// TIA Portal project "Proyectogrupal" (V15)

(* hardware
DEVICE "S7-1200 station_1"  S7-1200 Station
   slot 0: "Rack_0"  S7-1200 Rack  Rack  V1.0
   slot 1: "PLC_1"  CPU 1215C AC/DC/Rly  6ES7 215-1BG40-0XB0  V4.2
*)

// ===== PLC "PLC_1"  CPU 1215C AC/DC/Rly =====

VAR_GLOBAL   // PLC tag table "Tabla de variables estándar"
   "Etapa_0" AT %M200.0 : Bool;
   "Etapa_1" AT %M200.1 : Bool;
   "Etapa_2" AT %M200.2 : Bool;
   "Etapa_3" AT %M200.3 : Bool;
   "Etapa_4" AT %M200.4 : Bool;
   "Etapa_5" AT %M200.5 : Bool;
   "Etapa_80" AT %M50.0 : Bool;
   "Etapa_82" AT %M50.2 : Bool;
   "Selector" AT %I0.0 : Bool;
   "PM" AT %I0.1 : Bool;
   "PP" AT %I0.2 : Bool;
   "SH" AT %IW64 : Int;
   "P" AT %IW66 : Int;
   "PV" AT %Q0.0 : Bool;
   "PR" AT %Q0.1 : Bool;
   "Motor_ON" AT %Q0.2 : Bool;
   "Motor_LR" AT %Q0.3 : Bool;
   "Velocidad" AT %MD100 : Real;
   "H" AT %MD800 : Real;
   "AI" AT %QW64 : Int;
   "Clock_Byte" AT %MB0 : Byte;
   "Clock_10Hz" AT %M0.0 : Bool;
   "Clock_5Hz" AT %M0.1 : Bool;
   "Clock_2.5Hz" AT %M0.2 : Bool;
   "Clock_2Hz" AT %M0.3 : Bool;
   "Clock_1.25Hz" AT %M0.4 : Bool;
   "Clock_1Hz" AT %M0.5 : Bool;
   "Clock_0.625Hz" AT %M0.6 : Bool;
   "Clock_0.5Hz" AT %M0.7 : Bool;
   "System_Byte" AT %MB1 : Byte;
   "FirstScan" AT %M1.0 : Bool;
   "DiagStatusUpdate" AT %M1.1 : Bool;
   "AlwaysTRUE" AT %M1.2 : Bool;
   "AlwaysFALSE" AT %M1.3 : Bool;
   "A" AT %MD900 : Real;
   "B(SH)" AT %MD450 : Real;
   "C" AT %MD950 : Real;
   "D(P)" AT %MD475 : Real;
END_VAR

// folder: System blocks/Program resources

DATA_BLOCK "T1_"   // DB2
{ S7_Optimized_Access := 'TRUE' }
AUTHOR : Simatic
FAMILY : IEC
NAME : IEC_TMR
VERSION : 1.0
// stored: InstanceOfName IEC_TIMER
"IEC_TIMER"
BEGIN
END_DATA_BLOCK

// folder: (top level)

FUNCTION "Grafcet_Stop" : Void   // FC1, LAD
{ S7_Optimized_Access := 'TRUE' }
VERSION : 0.1
BEGIN

REGION Network 1
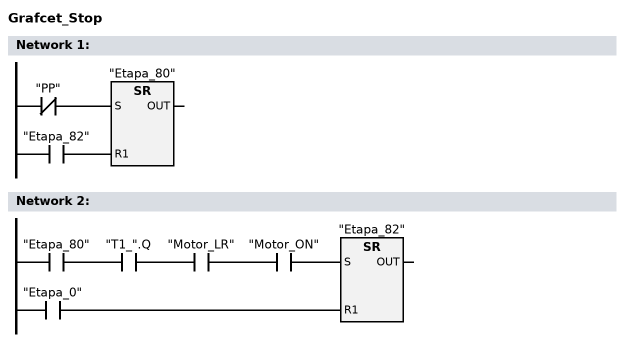
   RUNG wire#powerrail
      I_Contact( "PP" )
      S_SR(operand := "Etapa_80", r1 := wire#w1)
   END_RUNG
   RUNG wire#powerrail
      Contact( "Etapa_82" )
   END_RUNG wire#w1
   // the same network as SCL:
   IF NOT "PP" THEN
       "Etapa_80" := TRUE;   // SR flip-flop
   END_IF;
   IF "Etapa_82" THEN "Etapa_80" := FALSE; END_IF;
END_REGION

REGION Network 2
   RUNG wire#powerrail
      Contact( "Etapa_80" )
      Contact( "T1_".Q )
      Contact( "Motor_LR" )
      Contact( "Motor_ON" )
      S_SR(operand := "Etapa_82", r1 := wire#w1)
   END_RUNG
   RUNG wire#powerrail
      Contact( "Etapa_0" )
   END_RUNG wire#w1
   // the same network as SCL:
   IF "Etapa_80" AND "T1_".Q AND "Motor_LR" AND "Motor_ON" THEN
       "Etapa_82" := TRUE;   // SR flip-flop
   END_IF;
   IF "Etapa_0" THEN "Etapa_82" := FALSE; END_IF;
END_REGION
END_FUNCTION

FUNCTION "Grafcet_Automatico" : Void   // FC2, LAD
{ S7_Optimized_Access := 'TRUE' }
VERSION : 0.1
BEGIN

REGION Network 1
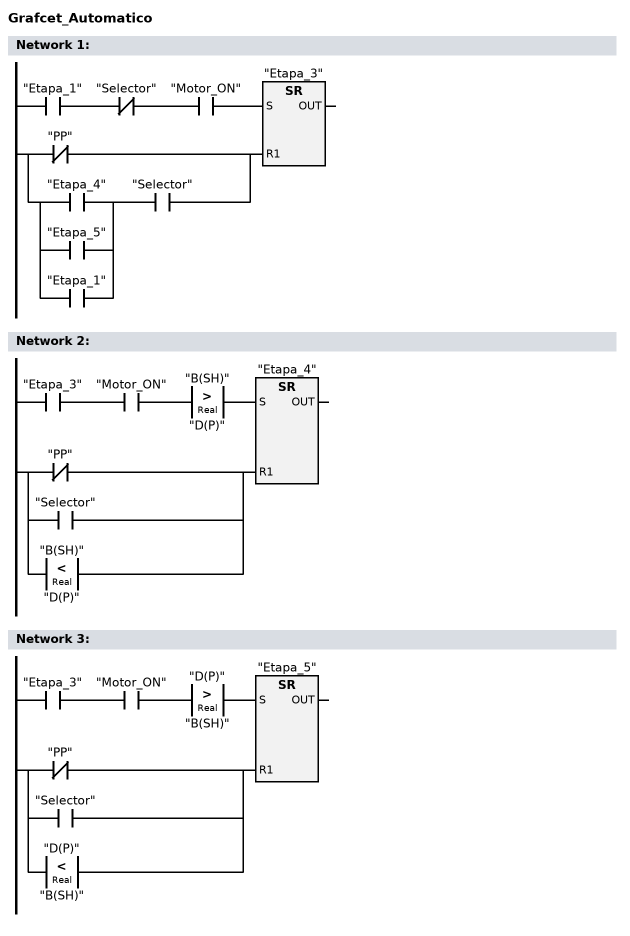
   RUNG wire#powerrail
      Contact( "Etapa_1" )
      I_Contact( "Selector" )
      Contact( "Motor_ON" )
      S_SR(operand := "Etapa_3", r1 := wire#w2)
   END_RUNG
   RUNG wire#powerrail
      I_Contact( "PP" )
   END_RUNG wire#w2
   RUNG wire#powerrail
      Contact( "Etapa_4" )
      wire#w1
      Contact( "Selector" )
   END_RUNG wire#w2
   RUNG wire#powerrail
      Contact( "Etapa_5" )
   END_RUNG wire#w1
   RUNG wire#powerrail
      Contact( "Etapa_1" )
   END_RUNG wire#w1
   // the same network as SCL:
   IF "Etapa_1" AND NOT "Selector" AND "Motor_ON" THEN
       "Etapa_3" := TRUE;   // SR flip-flop
   END_IF;
   IF NOT "PP" OR (("Etapa_4" OR "Etapa_5" OR "Etapa_1") AND "Selector") THEN "Etapa_3" := FALSE; END_IF;
END_REGION

REGION Network 2
   RUNG wire#powerrail
      Contact( "Etapa_3" )
      Contact( "Motor_ON" )
      { S7_Templates := "SrcType := Real" } GT_Contact(in1 := "B(SH)", in2 := "D(P)")
      S_SR(operand := "Etapa_4", r1 := wire#w1)
   END_RUNG
   RUNG wire#powerrail
      I_Contact( "PP" )
   END_RUNG wire#w1
   RUNG wire#powerrail
      Contact( "Selector" )
   END_RUNG wire#w1
   RUNG wire#powerrail
      { S7_Templates := "SrcType := Real" } LT_Contact(in1 := "B(SH)", in2 := "D(P)")
   END_RUNG wire#w1
   // the same network as SCL:
   IF "Etapa_3" AND "Motor_ON" AND ("B(SH)" > "D(P)") THEN
       "Etapa_4" := TRUE;   // SR flip-flop
   END_IF;
   IF NOT "PP" OR "Selector" OR ("B(SH)" < "D(P)") THEN "Etapa_4" := FALSE; END_IF;
END_REGION

REGION Network 3
   RUNG wire#powerrail
      Contact( "Etapa_3" )
      Contact( "Motor_ON" )
      { S7_Templates := "SrcType := Real" } GT_Contact(in1 := "D(P)", in2 := "B(SH)")
      S_SR(operand := "Etapa_5", r1 := wire#w1)
   END_RUNG
   RUNG wire#powerrail
      I_Contact( "PP" )
   END_RUNG wire#w1
   RUNG wire#powerrail
      Contact( "Selector" )
   END_RUNG wire#w1
   RUNG wire#powerrail
      { S7_Templates := "SrcType := Real" } LT_Contact(in1 := "D(P)", in2 := "B(SH)")
   END_RUNG wire#w1
   // the same network as SCL:
   IF "Etapa_3" AND "Motor_ON" AND ("D(P)" > "B(SH)") THEN
       "Etapa_5" := TRUE;   // SR flip-flop
   END_IF;
   IF NOT "PP" OR "Selector" OR ("D(P)" < "B(SH)") THEN "Etapa_5" := FALSE; END_IF;
END_REGION
END_FUNCTION

FUNCTION "Grafcet_Manual" : Void   // FC3, LAD
{ S7_Optimized_Access := 'TRUE' }
VERSION : 0.1
BEGIN

REGION Network 1
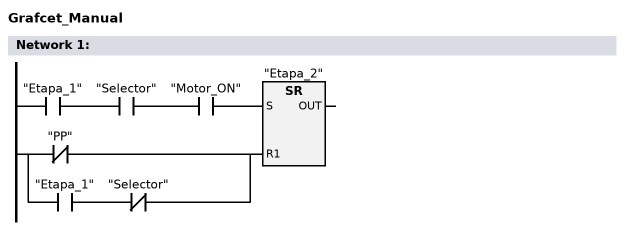
   RUNG wire#powerrail
      Contact( "Etapa_1" )
      Contact( "Selector" )
      Contact( "Motor_ON" )
      S_SR(operand := "Etapa_2", r1 := wire#w1)
   END_RUNG
   RUNG wire#powerrail
      I_Contact( "PP" )
   END_RUNG wire#w1
   RUNG wire#powerrail
      Contact( "Etapa_1" )
      I_Contact( "Selector" )
   END_RUNG wire#w1
   // the same network as SCL:
   IF "Etapa_1" AND "Selector" AND "Motor_ON" THEN
       "Etapa_2" := TRUE;   // SR flip-flop
   END_IF;
   IF NOT "PP" OR ("Etapa_1" AND NOT "Selector") THEN "Etapa_2" := FALSE; END_IF;
END_REGION
END_FUNCTION

FUNCTION "Grafcet_Acciones" : Void   // FC4, LAD
{ S7_Optimized_Access := 'TRUE' }
VERSION : 0.1
BEGIN

REGION Network 1
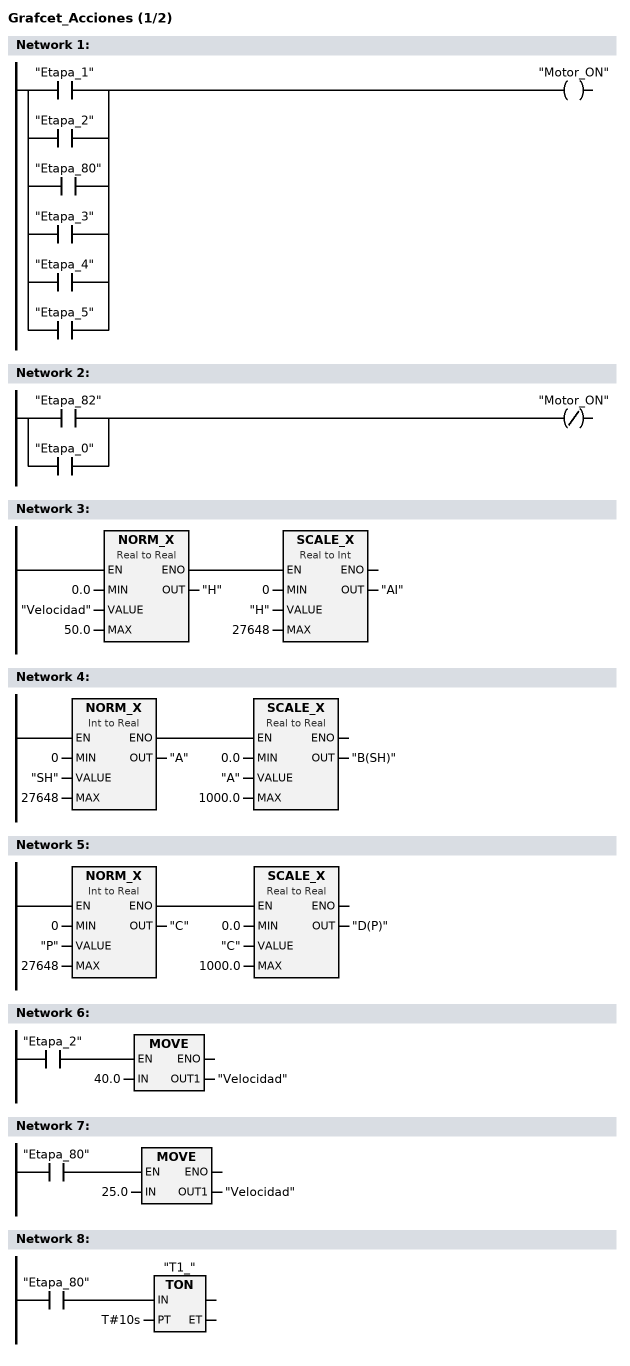
   RUNG wire#powerrail
      Contact( "Etapa_1" )
      wire#w1
      Coil( "Motor_ON" )
   END_RUNG
   RUNG wire#powerrail
      Contact( "Etapa_2" )
   END_RUNG wire#w1
   RUNG wire#powerrail
      Contact( "Etapa_80" )
   END_RUNG wire#w1
   RUNG wire#powerrail
      Contact( "Etapa_3" )
   END_RUNG wire#w1
   RUNG wire#powerrail
      Contact( "Etapa_4" )
   END_RUNG wire#w1
   RUNG wire#powerrail
      Contact( "Etapa_5" )
   END_RUNG wire#w1
   // the same network as SCL:
   "Motor_ON" := "Etapa_1" OR "Etapa_2" OR "Etapa_80" OR "Etapa_3" OR "Etapa_4" OR "Etapa_5";
END_REGION

REGION Network 2
   RUNG wire#powerrail
      Contact( "Etapa_82" )
      wire#w1
      I_Coil( "Motor_ON" )
   END_RUNG
   RUNG wire#powerrail
      Contact( "Etapa_0" )
   END_RUNG wire#w1
   // the same network as SCL:
   "Motor_ON" := NOT ("Etapa_82" OR "Etapa_0");
END_REGION

REGION Network 3
   RUNG wire#powerrail
      { S7_Templates := "[SrcType := Real, DestType := Real]" } Normalize(min := 0.0, value := "Velocidad", max := 50.0, out => "H")
      { S7_Templates := "[SrcType := Real, DestType := Int]" } Scale(min := 0, value := "H", max := 27648, out => "AI")
   END_RUNG
   // the same network as SCL:
   "H" := NORM_X(MIN := 0.0, VALUE := "Velocidad", MAX := 50.0);
   "AI" := SCALE_X(MIN := 0, VALUE := "H", MAX := 27648);
END_REGION

REGION Network 4
   RUNG wire#powerrail
      { S7_Templates := "[SrcType := Int, DestType := Real]" } Normalize(min := 0, value := "SH", max := 27648, out => "A")
      { S7_Templates := "[SrcType := Real, DestType := Real]" } Scale(min := 0.0, value := "A", max := 1000.0, out => "B(SH)")
   END_RUNG
   // the same network as SCL:
   "A" := NORM_X(MIN := 0, VALUE := "SH", MAX := 27648);
   "B(SH)" := SCALE_X(MIN := 0.0, VALUE := "A", MAX := 1000.0);
END_REGION

REGION Network 5
   RUNG wire#powerrail
      { S7_Templates := "[SrcType := Int, DestType := Real]" } Normalize(min := 0, value := "P", max := 27648, out => "C")
      { S7_Templates := "[SrcType := Real, DestType := Real]" } Scale(min := 0.0, value := "C", max := 1000.0, out => "D(P)")
   END_RUNG
   // the same network as SCL:
   "C" := NORM_X(MIN := 0, VALUE := "P", MAX := 27648);
   "D(P)" := SCALE_X(MIN := 0.0, VALUE := "C", MAX := 1000.0);
END_REGION

REGION Network 6
   RUNG wire#powerrail
      Contact( "Etapa_2" )
      Move(in := 40.0, out1 => "Velocidad")
   END_RUNG
   // the same network as SCL:
   IF "Etapa_2" THEN "Velocidad" := 40.0; END_IF;
END_REGION

REGION Network 7
   RUNG wire#powerrail
      Contact( "Etapa_80" )
      Move(in := 25.0, out1 => "Velocidad")
   END_RUNG
   // the same network as SCL:
   IF "Etapa_80" THEN "Velocidad" := 25.0; END_IF;
END_REGION

REGION Network 8
   "T1_".TON(IN := "Etapa_80", PT := T#10s);
END_REGION

REGION Network 9
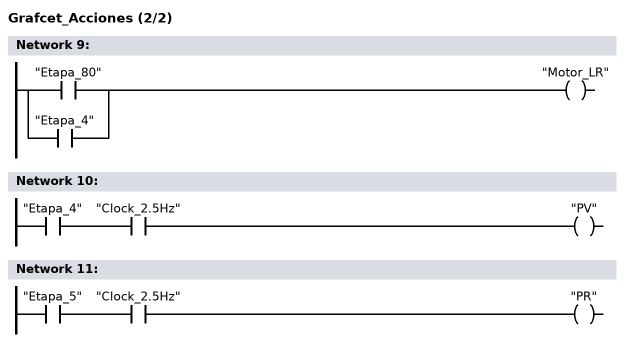
   RUNG wire#powerrail
      Contact( "Etapa_80" )
      wire#w1
      Coil( "Motor_LR" )
   END_RUNG
   RUNG wire#powerrail
      Contact( "Etapa_4" )
   END_RUNG wire#w1
   // the same network as SCL:
   "Motor_LR" := "Etapa_80" OR "Etapa_4";
END_REGION

REGION Network 10
   RUNG wire#powerrail
      Contact( "Etapa_4" )
      Contact( "Clock_2.5Hz" )
      Coil( "PV" )
   END_RUNG
   // the same network as SCL:
   "PV" := "Etapa_4" AND "Clock_2.5Hz";
END_REGION

REGION Network 11
   RUNG wire#powerrail
      Contact( "Etapa_5" )
      Contact( "Clock_2.5Hz" )
      Coil( "PR" )
   END_RUNG
   // the same network as SCL:
   "PR" := "Etapa_5" AND "Clock_2.5Hz";
END_REGION
END_FUNCTION

ORGANIZATION_BLOCK "Main"   // OB1, LAD, ProgramCycle
TITLE = "Main Program Sweep (Cycle)"
{ S7_Optimized_Access := 'TRUE' }
VERSION : 0.1
   VAR_INPUT
      Initial_Call : Bool;   // Initial call of this OB
      Remanence : Bool;   // =True, if remanent data are available
   END_VAR
BEGIN

REGION Network 1
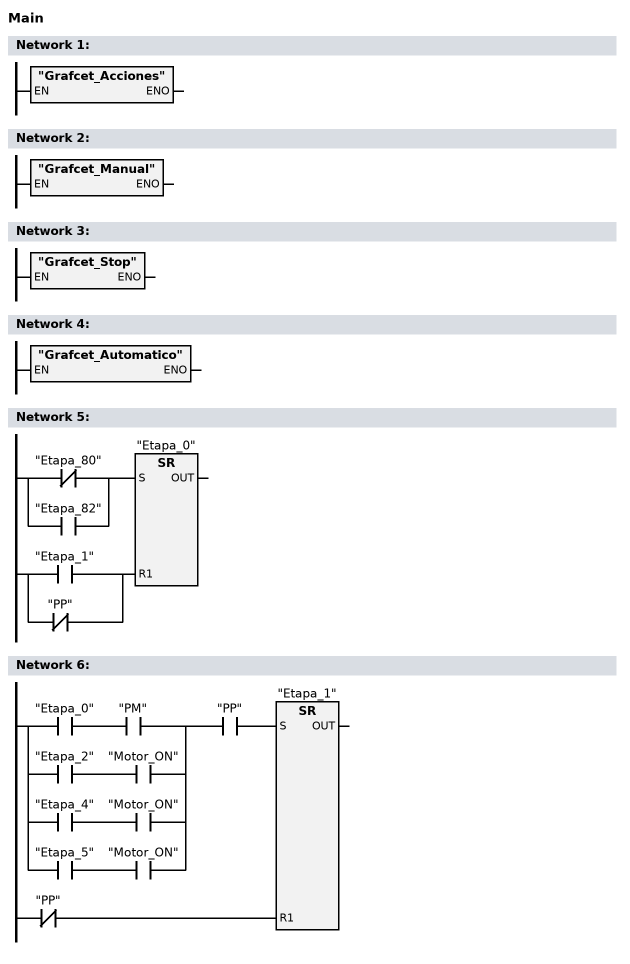
   RUNG wire#powerrail
      "Grafcet_Acciones"()
   END_RUNG
   // the same network as SCL:
   "Grafcet_Acciones"();
END_REGION

REGION Network 2
   RUNG wire#powerrail
      "Grafcet_Manual"()
   END_RUNG
   // the same network as SCL:
   "Grafcet_Manual"();
END_REGION

REGION Network 3
   RUNG wire#powerrail
      "Grafcet_Stop"()
   END_RUNG
   // the same network as SCL:
   "Grafcet_Stop"();
END_REGION

REGION Network 4
   RUNG wire#powerrail
      "Grafcet_Automatico"()
   END_RUNG
   // the same network as SCL:
   "Grafcet_Automatico"();
END_REGION

REGION Network 5
   RUNG wire#powerrail
      I_Contact( "Etapa_80" )
      wire#w1
      S_SR(operand := "Etapa_0", r1 := wire#w2)
   END_RUNG
   RUNG wire#powerrail
      Contact( "Etapa_82" )
   END_RUNG wire#w1
   RUNG wire#powerrail
      Contact( "Etapa_1" )
   END_RUNG wire#w2
   RUNG wire#powerrail
      I_Contact( "PP" )
   END_RUNG wire#w2
   // the same network as SCL:
   IF NOT "Etapa_80" OR "Etapa_82" THEN
       "Etapa_0" := TRUE;   // SR flip-flop
   END_IF;
   IF "Etapa_1" OR NOT "PP" THEN "Etapa_0" := FALSE; END_IF;
END_REGION

REGION Network 6
   RUNG wire#powerrail
      Contact( "Etapa_0" )
      Contact( "PM" )
      wire#w1
      Contact( "PP" )
      S_SR(operand := "Etapa_1", r1 := wire#w2)
   END_RUNG
   RUNG wire#powerrail
      Contact( "Etapa_2" )
      Contact( "Motor_ON" )
   END_RUNG wire#w1
   RUNG wire#powerrail
      Contact( "Etapa_4" )
      Contact( "Motor_ON" )
   END_RUNG wire#w1
   RUNG wire#powerrail
      Contact( "Etapa_5" )
      Contact( "Motor_ON" )
   END_RUNG wire#w1
   RUNG wire#powerrail
      I_Contact( "PP" )
   END_RUNG wire#w2
   // the same network as SCL:
   IF (("Etapa_0" AND "PM") OR ("Etapa_2" AND "Motor_ON") OR ("Etapa_4" AND "Motor_ON") OR ("Etapa_5" AND "Motor_ON")) AND "PP" THEN
       "Etapa_1" := TRUE;   // SR flip-flop
   END_IF;
   IF NOT "PP" THEN "Etapa_1" := FALSE; END_IF;
END_REGION
END_ORGANIZATION_BLOCK